FUNCTION_BLOCK CbVtStatus (* This function is called in case of every page change - you can do e. g. initialisations ... *)
  (* Standard: ISO 11783-6; Description: Copyright (c) 2022 HR Agrartechnik GmbH This program and the accompanying materials are made available under the terms of the Eclipse Public License 2.0 which is available at https://www.eclipse.org/legal/epl-2.0/ SPDX-License-Identifier: EPL-2.0 This function is called in case of every page change - you can do e. g. initialisations ... *)
  (* Version 1.0, 2022-07-20, Franz Höpfinger, HR Agrartechnik GmbH *)
  PACKAGE isobus::ut;
  IMPORT eclipse4diac::core::TypeHash;
  IMPORT isobus::ut::IDs::ID_NULL;
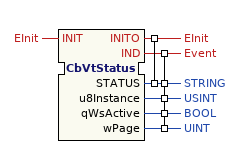
  EVENT_INPUT
    INIT : EInit; (* Service Initialization *)
  END_EVENT
  EVENT_OUTPUT
    INITO : EInit WITH STATUS; (* Initialization Confirm *)
    IND WITH STATUS, wPage, qWsActive, u8Instance; (* Indication from Resource *)
  END_EVENT
  VAR_OUTPUT
    STATUS : STRING; (* Service Status *)
    u8Instance : USINT; (* Identifier of the client instance *)
    qWsActive : BOOL; (* true, if the working set is active (displayed on screen) *)
    wPage : UINT := ID_NULL; (* Contains the object ID of the open/last mask, or NULL object ID if unknown (ID_NULL = 0xFFFF) *)
  END_VAR
END_FUNCTION_BLOCK
